(*
Registers component directly in declaration block. Alternative function: `RegComp`.
*)
FUNCTION_BLOCK Comp IMPLEMENTS I_Debug

//FB_Init is always available implicitly and it is used primarily for initialization.
//The return value is not evaluated. For a specific influence, you can also declare the
//methods explicitly and provide additional code there with the standard initialization
//code. You can evaluate the return value.
METHOD FB_Init: BOOL
VAR_INPUT
    bInitRetains: BOOL; // TRUE: the retain variables are initialized (reset warm / reset cold)
    bInCopyCode: BOOL;  // TRUE: the instance will be copied to the copy code afterward (online change)

	iComponent	: I_Component; // Component to register
	iEntity		: I_Entity; // Component owner
END_VAR
VAR
	_nResult	: Result;
END_VAR
IF IsErr(_RegComp(iEntity, iComponent), nOut => _nResult) THEN
	DebugMsg(THIS^, Tc2_Standard.CONCAT('Failed with code: ', ResultToStr(_nResult)));
END_IF
END_METHOD

END_FUNCTION_BLOCK

(* stored: Version 1.1.0.1
   POU Comp: Id {3b4f07cd-ce06-44c8-8976-14381e17260e}, SpecialFunc None
   Method Fb_init: Id {735d5726-36c2-48ac-a9f6-84bea416f22a} *)
